FUNCTION_BLOCK PUBLIC VelocityCtrlAxis_FB
VAR_INPUT
	
	rAxisBasicFB 		: REFERENCE TO BasicAxis_FB ;
	rVelocityCtrl	 	: REFERENCE TO VelocityCtrl_typ ;
		
END_VAR

VAR_OUTPUT
END_VAR
	
VAR
	LogMsgInit		: BOOL;
	LogMsg_0 		: LogMsg ;
	
//	GetCycleTime:	FB_CTRL_GET_TASK_CYCLETIME;
//	CycleTime:		TIME;
//	CycleTimeInit:	BOOL;
	
	
	fbGetCurTaskIdx: 		GETCURTASKINDEX;
    TaskCycleTimeUDINT: 	UDINT;
    TaskCycleTime: 			TIME;

	EnableTrigger : Trigger ;
	
	DisableTriger	: Trigger ;
	Disable			: BOOL ;
	
// Change Oper params
	ChangeModeTrigger   : Trigger ;
	CngToVelocityState 	: SINT;
	PrevCngToVelocityState : SINT;
	// Change Oper params
	InitSctrlTrigger : Trigger ;
	InitSctrlState 	 : SINT;	

	
	ErrorTrig : Trigger ;
	AxisStep     : eVelocityCtrlState ;
	ReturnToAxisStep     : eVelocityCtrlState ;
	
	LastAxisStep : eVelocityCtrlState ;
	
	tmp_ErrorEntry			: Eh_ErrorEntry_typ;
	
	
	
	ReadPosCtrlParamDone 	: BOOL;	
	OldCyclicTorque 		: LREAL;		
	OldSctrlKp 				: LREAL;
	OldSctrlKi 				: LREAL;
	PrevVel 				: LREAL;
	Error					: BOOL;
	//Paramter
		
	CyclicTorqueAtPositionCtrl : LREAL;	
	

	
	Delay 			:	 TON;
	
	StartTestRead: BOOL;
	TestRead : BOOL;
END_VAR

// 
// At default set default torque
//
// Change mode to velocity control
// 
//
//
//
//
IF __ISVALIDREF( rAxisBasicFB) AND __ISVALIDREF(rVelocityCtrl) THEN
	
	

IF NOT LogMsgInit THEN 
	LogMsg_0.logData.category:=	rAxisBasicFB.AxisCtrlPtr^.Input.Parameter.ThreadName;     
	LogMsg_0.Enable:= 	TRUE; 	
END_IF

IF (TaskCycleTimeUDINT = 0) THEN
	fbGetCurTaskIdx();
	TaskCycleTimeUDINT := _TaskInfo[fbGetCurTaskIdx.index].CycleTime;
	TaskCycleTime	:= UDINT_TO_TIME(TaskCycleTimeUDINT/10000); 
END_IF



LogMsg_0.ptrGlobalArray:= 	ADR(LogGlobalArray);
LogMsg_0.ptrEncoderAngle:= 	ADR(rAxisBasicFB.AxisCtrlPtr^.Input.Parameter.PosForLog);



//in case of Stop go to STATE_WAIT
IF (rVelocityCtrl.Output.Status.Active)AND(NOT rVelocityCtrl.Output.Status.InStopVelCtrl)  THEN
	
	
	IF rAxisBasicFB.AxisCtrlPtr^.Output.Status.FAULT THEN
 
			AxisStep := eVelocityCtrlState.VELOCITY_CTRL_STATE_ERROR;	

	ELSIF (rAxisBasicFB.AxisCtrlPtr^.Input.Command.Halt) OR rVelocityCtrl.Input.Command.Stop THEN
		rVelocityCtrl.Input.Command.Stop := FALSE;
		Meth_stop(FALSE);
		AxisStep := eVelocityCtrlState.VELOCITY_CTRL_STATE_STOP ;

		
	ELSIF (rAxisBasicFB.AxisCtrlPtr^.Input.Command.Stop)  THEN 
		AxisStep := eVelocityCtrlState.VELOCITY_CTRL_ACTIVE_STAND_STILL;
		PrevVel :=  rVelocityCtrl.Input.Parameter.CyclicVelocity := 0;
	END_IF	
	
END_IF


IF EnableTrigger.EDGEPOS(rVelocityCtrl.Input.Command.Enable) THEN
 	IF (NOT rVelocityCtrl.Output.Status.Active) AND AxisStep = eVelocityCtrlState.VELOCITY_CTRL_STATE_READY THEN
		METH_ChangeToVelMode(FALSE);
		AxisStep := VELOCITY_CTRL_CNG_TO_VEL_MODE ;
	END_IF	
		
END_IF		
	
IF EnableTrigger.EDGENEG( rVelocityCtrl.Input.Command.Enable) THEN
	IF (rVelocityCtrl.Output.Status.Active) THEN
 		Meth_ExitVelCtrl(FALSE);
		AxisStep :=  eVelocityCtrlState.VELOCITY_CTRL_DISABLE;
	END_IF	
	
END_IF		



CASE AxisStep OF
		
	(******************** WAIT *************************)
		
	VELOCITY_CTRL_STATE_WAIT:	
		rVelocityCtrl.Output.Status.Active := FALSE;
		IF rAxisBasicFB.AxisCtrlPtr^.Output.Status.AxisInitDone
			 THEN
			AxisStep := VELOCITY_CTRL_STATE_READY ;
		END_IF
		
		THIS^.ResetAll_MC_FB();
		
	VELOCITY_CTRL_STATE_READY:
	
		rVelocityCtrl.Output.Status.Active := FALSE;
		IF rVelocityCtrl.Input.Command.InitSctrl THEN
				
				rVelocityCtrl.Input.Command.InitSctrl := FALSE;
				rVelocityCtrl.Output.Status.SctrlInitialized := FALSE;
				Meth_InitSctrl(FALSE);
				
				rAxisBasicFB.Meth_WriteObj(FALSE,enumMotionObject.VEL_KI,0);
				AxisStep :=VELOCITY_CTRL_InitSctrl;
				ReturnToAxisStep := VELOCITY_CTRL_STATE_READY;
 								
		ELSIF rVelocityCtrl.Input.Command.Stop THEN
			
			rVelocityCtrl.Input.Command.Stop  := FALSE;
			AxisStep := VELOCITY_CTRL_STATE_STOP ;
			
		ELSIF rVelocityCtrl.Input.Parameter.CyclicTorque <> OldCyclicTorque THEN
				
				Error := FALSE;
				ReturnToAxisStep := VELOCITY_CTRL_STATE_READY;
				AxisStep :=VELOCITY_CTRL_CHANGE_TORQUE;
				
				rAxisBasicFB.Meth_CngTorqueOffset(FALSE,0);
				rAxisBasicFB.Meth_CngMaxTorque(FALSE,0);
				ReturnToAxisStep := VELOCITY_CTRL_STATE_READY;
				rAxisBasicFB.Meth_WriteObj(FALSE,enumMotionObject.VEL_KI,0);	
				rVelocityCtrl.Output.Status.UpdateTorqueDone := FALSE;		
		END_IF
		

//ReadPosCtrlParamDone
		
	VELOCITY_CTRL_CNG_TO_VEL_MODE:
		// Change mode to velocity control
		IF METH_ChangeToVelMode(TRUE) THEN
			rVelocityCtrl.Output.Status.Active := TRUE;
			AxisStep :=VELOCITY_CTRL_MOVE_VELOCITY;
		END_IF	
			
	VELOCITY_CTRL_READ_POS_CTRL_VALUES:
			IF Meth_ReadPosCtrlValues(TRUE) THEN
				AxisStep :=VELOCITY_CTRL_MOVE_VELOCITY;
			END_IF
	
				
	VELOCITY_CTRL_MOVE_VELOCITY:
	
		IF rVelocityCtrl.Input.Parameter.CyclicVelocity <>0 OR rAxisBasicFB.AxisCtrlPtr^.Output.monitor.ActVelocity <>0  THEN
			Meth_MoveVel();
			AxisStep := VELOCITY_CTRL_WAIT_MOVE_VELOCITY_DONE;
		ELSE
			AxisStep := VELOCITY_CTRL_ACTIVE;
		END_IF	
	
	
	VELOCITY_CTRL_WAIT_MOVE_VELOCITY_DONE:	
		IF rAxisBasicFB.AxisCtrlPtr^.Output.Status.MC_MoveVelocity.In_Velocity THEN
			IF rVelocityCtrl.Input.Parameter.CyclicTorque <> 0 THEN
				Error := FALSE;
				ReturnToAxisStep := VELOCITY_CTRL_ACTIVE;
				AxisStep :=VELOCITY_CTRL_CHANGE_TORQUE;
				rAxisBasicFB.Meth_CngTorqueOffset(FALSE,0);
				rAxisBasicFB.Meth_CngMaxTorque(FALSE,0);
				ReturnToAxisStep := VELOCITY_CTRL_ACTIVE;
				rAxisBasicFB.Meth_WriteObj(FALSE,enumMotionObject.VEL_KI,0);
			ELSE
				PrevVel := rVelocityCtrl.Input.Parameter.CyclicVelocity;
				AxisStep := VELOCITY_CTRL_ACTIVE;
			END_IF	 
	END_IF
		
		
	VELOCITY_CTRL_ACTIVE:
	
			rVelocityCtrl.Output.Status.Active := TRUE;
			IF rVelocityCtrl.Input.Command.Stop THEN
				meth_Stop(FALSE);
				rVelocityCtrl.Input.Command.Stop  := FALSE;
				AxisStep := VELOCITY_CTRL_STATE_STOP ;
				
			ELSIF rVelocityCtrl.Input.Command.InitSctrl THEN
				
				rVelocityCtrl.Input.Command.InitSctrl := FALSE;
				rVelocityCtrl.Output.Status.SctrlInitialized := FALSE;
				Meth_InitSctrl(FALSE);
				
				rAxisBasicFB.Meth_WriteObj(FALSE,enumMotionObject.VEL_KI,0);
				AxisStep :=VELOCITY_CTRL_InitSctrl;
				ReturnToAxisStep := VELOCITY_CTRL_ACTIVE;
				
			ELSIF rVelocityCtrl.Input.Parameter.CyclicTorque <> OldCyclicTorque THEN
				
				Error := FALSE;
				ReturnToAxisStep := VELOCITY_CTRL_ACTIVE;
				AxisStep :=VELOCITY_CTRL_CHANGE_TORQUE;
				rAxisBasicFB.Meth_CngTorqueOffset(FALSE,0);
				rAxisBasicFB.Meth_CngMaxTorque(FALSE,0);
				ReturnToAxisStep := VELOCITY_CTRL_ACTIVE;
				rAxisBasicFB.Meth_WriteObj(FALSE,enumMotionObject.VEL_KI,0);				
			ELSIF rVelocityCtrl.Input.Parameter.CyclicVelocity <> rAxisBasicFB.AxisCtrlPtr^.Input.Parameter.Velocity THEN
					AxisStep := VELOCITY_CTRL_MOVE_VELOCITY;
		 	
			ELSIF rVelocityCtrl.Input.Parameter.CyclicVelocity <> PrevVel THEN
				
				AxisStep := VELOCITY_CTRL_MOVE_VELOCITY;
				
			END_IF	
			
	VELOCITY_CTRL_ACTIVE_STAND_STILL:
			rVelocityCtrl.Output.Status.Active := TRUE;
 			
			IF rVelocityCtrl.Input.Parameter.CyclicVelocity <> PrevVel THEN
				
				AxisStep := VELOCITY_CTRL_MOVE_VELOCITY;
			
			
			ELSIF rVelocityCtrl.Input.Command.InitSctrl THEN
				
				rVelocityCtrl.Input.Command.InitSctrl := FALSE;
				rVelocityCtrl.Output.Status.SctrlInitialized := FALSE;
				Meth_InitSctrl(FALSE);
				
				rAxisBasicFB.Meth_WriteObj(FALSE,enumMotionObject.VEL_KI,0);
				AxisStep :=VELOCITY_CTRL_InitSctrl;
				ReturnToAxisStep := VELOCITY_CTRL_ACTIVE_STAND_STILL;
				
			ELSIF rVelocityCtrl.Input.Parameter.CyclicTorque <> OldCyclicTorque THEN
				
				Error := FALSE;
				ReturnToAxisStep := VELOCITY_CTRL_ACTIVE;
				AxisStep :=VELOCITY_CTRL_CHANGE_TORQUE;
				rAxisBasicFB.Meth_CngTorqueOffset(FALSE,0);
				rAxisBasicFB.Meth_CngMaxTorque(FALSE,0);
				ReturnToAxisStep := VELOCITY_CTRL_ACTIVE_STAND_STILL;
				rAxisBasicFB.Meth_WriteObj(FALSE,enumMotionObject.VEL_KI,0);

		 	
			ELSIF rAxisBasicFB.AxisCtrlPtr^.Output.Status.AxisStatus.Coupled THEN
				IF rAxisBasicFB.AxisCtrlPtr^.Output.monitor.ActVelocity <> 0 THEN
					AxisStep := VELOCITY_CTRL_ACTIVE;
				END_IF 
			END_IF	

	VELOCITY_CTRL_InitSctrl:
	
			IF Meth_InitSctrl(TRUE,Error=>Error) THEN
				AxisStep :=ReturnToAxisStep;			
			END_IF
			
			IF Error THEN
			//	
			END_IF
	VELOCITY_CTRL_CHANGE_TORQUE:	
				
			IF rVelocityCtrl.Input.Parameter.TorqueMode = eTorqueMode.mcFF THEN
				//IF rAxisBasicFB.Meth_CngTorqueOffset(TRUE,rVelocityCtrl.Input.Parameter.CyclicTorque, Error => Error ) THEN
				IF  rAxisBasicFB.Meth_WriteObj(TRUE, enumMotionObject.TORQUE_OFFSET,rVelocityCtrl.Input.Parameter.CyclicTorque, Error => Error ) THEN
					fnLogMsg(ADR(LogMsg_0),LOG_INFO,'Vel Ctrl Change Torque to=%d',LREAL_TO_DINT(rVelocityCtrl.Input.Parameter.CyclicTorque*1000),0,0);
					
					OldCyclicTorque := rVelocityCtrl.Input.Parameter.CyclicTorque;
					rAxisBasicFB.Meth_CngTorqueOffset(FALSE,rVelocityCtrl.Input.Parameter.CyclicTorque);
					AxisStep :=ReturnToAxisStep;	
					rVelocityCtrl.Output.monitor.SetCyclicTorque := rVelocityCtrl.Input.Parameter.CyclicTorque ;
				END_IF							
			
			ELSIF rVelocityCtrl.Input.Parameter.TorqueMode = eTorqueMode.mcLimit THEN
				//IF rAxisBasicFB.Meth_CngMaxTorque(TRUE,rVelocityCtrl.Input.Parameter.CyclicTorque , Error => Error) THEN
				IF  rAxisBasicFB.Meth_WriteObj(TRUE, enumMotionObject.MAX_TORQUE,rVelocityCtrl.Input.Parameter.CyclicTorque, Error => Error ) THEN					
					OldCyclicTorque := rVelocityCtrl.Input.Parameter.CyclicTorque;
					rVelocityCtrl.Output.monitor.SetCyclicTorque := rVelocityCtrl.Input.Parameter.CyclicTorque ;
					rVelocityCtrl.Output.Status.UpdateTorqueDone := TRUE;
					AxisStep :=ReturnToAxisStep;
	
				END_IF
			END_IF
			
	eVelocityCtrlState.VELOCITY_CTRL_STATE_STOP:
		IF Meth_stop(TRUE) THEN
			
			PrevVel :=  rVelocityCtrl.Input.Parameter.CyclicVelocity := 0;
			AxisStep := eVelocityCtrlState.VELOCITY_CTRL_ACTIVE_STAND_STILL;
		END_IF
	
	
	eVelocityCtrlState.VELOCITY_CTRL_DISABLE:
		rVelocityCtrl.Output.Status.InStopVelCtrl := TRUE;
		IF Meth_ExitVelCtrl(TRUE) THEN
			rVelocityCtrl.Output.Status.InStopVelCtrl := FALSE;
			AxisStep := eVelocityCtrlState.VELOCITY_CTRL_STATE_READY;
		END_IF
	eVelocityCtrlState.VELOCITY_CTRL_STATE_RETURN_ORG_VALUES:
		IF Meth_ReturnOrgPosCtrlValues(TRUE) THEN				
			AxisStep := ReturnToAxisStep ;
		END_IF
		
	eVelocityCtrlState.VELOCITY_CTRL_STATE_ERROR:
			rVelocityCtrl.Output.Status.InStopVelCtrl := TRUE;
			IF Meth_ExitVelCtrl(TRUE) THEN			
				rVelocityCtrl.Output.Status.InStopVelCtrl := FALSE;
				AxisStep := eVelocityCtrlState.VELOCITY_CTRL_STATE_WAIT;
			END_IF

			

	
	
END_CASE 



//=====================================================================================================================\\

//IF CyclicAxisCtrlPtr^.Output.Error.ErrorID <> 0 THEN		
	//BasicAxisCtrlPtr^.Output.Error.ErrorID := CyclicAxisCtrlPtr^.Output.Error.ErrorID ;
	//CyclicAxisCtrlPtr^.Output.Error.ErrorID := 0;
//END_IF

	IF LastAxisStep <> AxisStep THEN
		
		fnLogMsg(ADR(LogMsg_0),LOG_INFO,'Vel Ctrl CurSt=%d LstSt=%d',AxisStep,LastAxisStep,0);
		LastAxisStep := AxisStep ;
	END_IF	
	
	IF StartTestRead THEN
		StartTestRead := FALSE;
		Meth_ReadPosCtrlValues(FALSE);
		TestRead := TRUE;
		
	ELSIF TestRead THEN
		IF Meth_ReadPosCtrlValues(TRUE) THEN
			TestRead := FALSE;
		END_IF	
		
	END_IF

	
	
//fnLogTransfer FUNCTION call
fnLogTransfer(ADR(LogMsg_0));
		

END_IF

METHOD AddNCError : BOOL
VAR_INPUT
	ErrorId			: UDINT;
	ErrorPrefix     : STRING[100];
END_VAR

	tmp_ErrorEntry.ErrorId		:= ErrorId;

	tmp_ErrorEntry.ErrorText	:= ErrorPrefix;

	tmp_ErrorEntry.ErrorText	:= CONCAT(tmp_ErrorEntry.ErrorText, UDINT_TO_STRING(tmp_ErrorEntry.ErrorId));
	tmp_ErrorEntry.ErrorText	:= CONCAT(tmp_ErrorEntry.ErrorText, 'Task: ');
	tmp_ErrorEntry.ErrorText	:= CONCAT(tmp_ErrorEntry.ErrorText, rVelocityCtrl.Input.Parameter.ThreadName);	
	tmp_ErrorEntry.ErrorText	:= CONCAT(tmp_ErrorEntry.ErrorText, FC_NcErrorMsg(tmp_ErrorEntry.ErrorId));	
	fnLogMsg(ADR(LogMsg_0),LOG_ERROR,tmp_ErrorEntry.ErrorText,0,0,0);	
	
	tmp_ErrorEntry.MotorEvents := CreateNCErrMsgDetails(tmp_ErrorEntry.ErrorId);
	
	rAxisBasicFB.AxisCtrlPtr^.Output.Error.fbErrorHandler.ErrorPush(tmp_ErrorEntry);
END_METHOD

METHOD METH_ChangeToVelMode : BOOL
VAR_INPUT
	Execute : BOOL;
END_VAR
VAR_INST
	DelayBeforeChangimeMode: TON;
END_VAR
IF InitSctrlTrigger.EDGEPOS( Execute) THEN
	CngToVelocityState := 1;
	METH_ChangeToVelMode := FALSE;
	rAxisBasicFB.AxisCtrlPtr^.Input.Command.Power := FALSE;
	
	OldCyclicTorque := 0;		
	OldSctrlKp 		:= 0;
	OldSctrlKi 		:= 0;			
	rAxisBasicFB.Meth_WriteObj (FALSE, enumMotionobject.OPERATION_MODE,DINT_TO_LREAL(eDriveModeOfOperation.CyclicSyncVelocity));

END_IF

IF InitSctrlTrigger.EDGENEG( Execute) THEN
	CngToVelocityState := 0;
END_IF


CASE CngToVelocityState OF
	0:
		METH_ChangeToVelMode := FALSE;
		 
	1:
		DelayBeforeChangimeMode.IN := FALSE;
		IF ReadPosCtrlParamDone = FALSE THEN
			 Meth_ReadPosCtrlValues(FALSE);
			 CngToVelocityState := CngToVelocityState +1;	
		ELSE
			CngToVelocityState := CngToVelocityState +2;
		END_IF		
	2:
		IF Meth_ReadPosCtrlValues(TRUE) THEN
			
			rAxisBasicFB.Meth_WriteObj (FALSE, enumMotionobject.OPERATION_MODE,eDriveModeOfOperation.CyclicSyncVelocity);
			
			CngToVelocityState := CngToVelocityState +1;
			
		END_IF
	3:	//Change mode to velocity control
		IF rAxisBasicFB.Meth_WriteObj (TRUE, enumMotionobject.OPERATION_MODE,eDriveModeOfOperation.CyclicSyncVelocity) THEN			
			rAxisBasicFB.Meth_WriteObj (FALSE, enumMotionobject.OPERATION_MODE,eDriveModeOfOperation.CyclicSyncVelocity);
			CngToVelocityState := CngToVelocityState +1;
		END_IF
		
	4://Disable Gain Control
		IF NOT rAxisBasicFB.AxisCtrlPtr^.Output.Status.MC_Power.Status THEN
			IF rAxisBasicFB.Meth_WriteObj (TRUE, enumMotionobject.GAIN_SCHEDULE,0) THEN			
				rAxisBasicFB.Meth_WriteObj (FALSE, enumMotionobject.OPERATION_MODE,eDriveModeOfOperation.CyclicSyncVelocity);			
				CngToVelocityState := CngToVelocityState +1;
			END_IF
		END_IF	
	
	5:	
		DelayBeforeChangimeMode.IN := TRUE;
		DelayBeforeChangimeMode.PT := T#10S;
		IF DelayBeforeChangimeMode.Q THEN
			rAxisBasicFB.AxisCtrlPtr^.Input.Command.Power := TRUE;
			IF rAxisBasicFB.AxisCtrlPtr^.Output.Status.AxisStatus.StandStill THEN
				CngToVelocityState := CngToVelocityState +1;
			END_IF
		END_IF	
	6:
		IF  rAxisBasicFB.Meth_WriteObj(TRUE, enumMotionObject.ACC_CLOSE_POS_ERR ,   rVelocityCtrl.Input.Parameter.CyclicVelocity    , Error =>Error ) THEN
			rAxisBasicFB.Meth_WriteObj(FALSE, enumMotionObject.ACC_CLOSE_POS_ERR ,0 );
			CngToVelocityState := CngToVelocityState +1;
		END_IF	
	
	7:	
		METH_ChangeToVelMode := TRUE;
END_CASE

DelayBeforeChangimeMode();

	IF CngToVelocityState <> PrevCngToVelocityState THEN
		
		fnLogMsg(ADR(LogMsg_0),LOG_INFO,'CngToVelocityState CurSt=%d LstSt=%d',CngToVelocityState,PrevCngToVelocityState,0);
		PrevCngToVelocityState := CngToVelocityState ;
	END_IF
END_METHOD

METHOD Meth_ExitVelCtrl : BOOL
VAR_INPUT
	Execute   : BOOL;
END_VAR

VAR_INST
	// Service Functions Variablea
	StopTrigger : Trigger ;
	ExitState  		 : SINT;
	PrevExitState   : SINT;
END_VAR

VAR_OUTPUT
	Error : BOOL;
END_VAR

IF StopTrigger.EDGEPOS(Execute) THEN
	ExitState  := 1;
	Meth_ExitVelCtrl := FALSE;
 	Meth_ReturnOrgPosCtrlValues(FALSE) ;
	Error := FALSE;
END_IF


IF StopTrigger.EDGENEG(Execute) THEN
	 PrevExitState := 0;
	 ExitState:= 0;
END_IF


CASE ExitState OF
	 		
	
	1:	 
		
//			
 //  	
		Delay(IN:=	FALSE);
		IF rAxisBasicFB.AxisCtrlPtr^.Output.Status.AxisStatus.StandStill = FALSE  AND rAxisBasicFB.AxisCtrlPtr^.Output.Status.AxisStatus.Disabled = FALSE THEN
		//	rAxisBasicFB.AxisCtrlPtr^.Input.Command.MoveVelocity := TRUE;	
		//	rAxisBasicFB.AxisCtrlPtr^.Input.Parameter.Velocity   := 100;
			rAxisBasicFB.AxisCtrlPtr^.Input.Command.Stop := TRUE;		
			ExitState := ExitState +1;
		ELSE
			ExitState := 3;
		END_IF	
					
   						
		
		
		
	2:
			IF (rAxisBasicFB.AxisCtrlPtr^.Output.Status.AxisStatus.StandStill OR rAxisBasicFB.AxisCtrlPtr^.Output.Status.AxisStatus.Disabled)				
			//IF rAxisBasicFB.AxisCtrlPtr^.Output.Status.MC_MoveVelocity.In_Velocity 
				 THEN
				Delay.PT := T#2S;
				Delay(IN:=	TRUE);
				IF Delay.Q THEN
					ExitState := ExitState +1;
				END_IF								
			END_IF

	
	3:
			rAxisBasicFB.AxisCtrlPtr^.Input.Command.Power := FALSE;

			ExitState := ExitState +1;

	4:
		IF rAxisBasicFB.AxisCtrlPtr^.Output.Status.AxisStatus.Disabled THEN
			IF ReadPosCtrlParamDone THEN
				IF  rAxisBasicFB.Meth_WriteObj(TRUE, enumMotionObject.ACC_CLOSE_POS_ERR ,  rVelocityCtrl.Output.monitor.OrgAccToCloseThePosError, Error =>Error ) THEN
					rAxisBasicFB.Meth_WriteObj(FALSE, enumMotionObject.ACC_CLOSE_POS_ERR ,0 );
					ExitState := ExitState +1;
				END_IF
			ELSE	
				ExitState := ExitState +1;
			END_IF
			
		END_IF	
	

	5:
		IF ReadPosCtrlParamDone THEN
			IF Meth_ReturnOrgPosCtrlValues(TRUE) THEN
				ExitState := ExitState +1;
			END_IF
		ELSE	
			ExitState := ExitState +1;
		END_IF
	
	
	6:		
		IF rAxisBasicFB.Meth_WriteObj (TRUE, enumMotionobject.OPERATION_MODE,TO_LREAL(eDriveModeOfOperation.CyclicSyncMode)) THEN
			rAxisBasicFB.Meth_WriteObj (FALSE, enumMotionobject.OPERATION_MODE,0);
			Delay.IN := FALSE;
			ExitState := ExitState +1;
		END_IF
	7:
			Delay.IN := TRUE;
			Delay.PT := T#2S;
			Delay();
			IF Delay.Q THEN
				ExitState := ExitState +1;
				Delay.IN := FALSE;
			END_IF

	8:
 		Meth_ExitVelCtrl := TRUE;
		

	

END_CASE

	IF ExitState <> PrevExitState THEN
		
		fnLogMsg(ADR(LogMsg_0),LOG_INFO,'Exit Vel Ctrl CurSt=%d LstSt=%d',ExitState,PrevExitState,0);
		PrevExitState := ExitState ;
	END_IF
END_METHOD

METHOD Meth_InitSctrl : BOOL
VAR_INPUT
	Execute : BOOL;
END_VAR


VAR_OUTPUT
	Error : BOOL;
END_VAR
IF InitSctrlTrigger.EDGEPOS(Execute) THEN
	InitSctrlState  := 1;
	Meth_InitSctrl := FALSE;
	rAxisBasicFB.Meth_InitVelKP (FALSE,0);
	rAxisBasicFB.Meth_InitVelKI(FALSE,0);
	Error := FALSE;
END_IF


IF InitSctrlTrigger.EDGENEG(Execute) THEN
	
	 InitSctrlState:= 0;
END_IF


CASE InitSctrlState OF
	 
		
	1:
		 			
			IF rAxisBasicFB.Meth_InitVelKP (TRUE,(rVelocityCtrl.Input.Parameter.SctrlKp), Error=>Error) THEN
				OldSctrlKp := rVelocityCtrl.Input.Parameter.SctrlKp;
				InitSctrlState := InitSctrlState +1;
				rAxisBasicFB.Meth_InitVelKP (FALSE,rVelocityCtrl.Input.Parameter.SctrlKp);
			END_IF	
  
			

	2:
	
		IF rAxisBasicFB.Meth_InitVelKI(TRUE,(rVelocityCtrl.Input.Parameter.SctrlKi), Error=>Error) THEN
			rAxisBasicFB.Meth_InitVelKP (FALSE,rVelocityCtrl.Input.Parameter.SctrlKi);
			OldSctrlKi := rVelocityCtrl.Input.Parameter.SctrlKi ;
			InitSctrlState := InitSctrlState +1;
		END_IF	

		IF Error THEN
		//	
		END_IF
		
	3:		
		rAxisBasicFB.Meth_WriteObj(FALSE,enumMotionObject.VEL_KI,0);
		rVelocityCtrl.Output.Status.SctrlInitialized := TRUE;
		Meth_InitSctrl := TRUE; 
	END_CASE
END_METHOD

METHOD Meth_MoveVel : BOOL
VAR_INPUT
END_VAR
	rAxisBasicFB.AxisCtrlPtr^.Input.Parameter.Velocity 	   := rVelocityCtrl.Input.Parameter.CyclicVelocity;
	rAxisBasicFB.AxisCtrlPtr^.Input.Parameter.Acceleration := rVelocityCtrl.Input.Parameter.Acceleration;
	rAxisBasicFB.AxisCtrlPtr^.Input.Parameter.Deceleration := rVelocityCtrl.Input.Parameter.Deceleration;
	
	rAxisBasicFB.AxisCtrlPtr^.Input.Command.MoveVelocity := TRUE;
END_METHOD

METHOD Meth_ReadPosCtrlValues : BOOL
VAR_INPUT
	Execute : BOOL;
END_VAR


VAR_INST
	// Service Functions Variablea
		 
	ReadOrginalValuesTrigger : Trigger ;
	ReadOrginalValuesState   : SINT;
END_VAR	

VAR_OUTPUT
	Error : BOOL;	
END_VAR
IF ReadOrginalValuesTrigger.EDGEPOS(Execute) THEN
	ReadOrginalValuesState  := 1;
	Meth_ReadPosCtrlValues := FALSE;
	Error := FALSE;
	rAxisBasicFB.Meth_ReadObj(FALSE, enumMotionObject.MAX_TORQUE, Value =>rVelocityCtrl.Output.monitor.OrgMaxTorque, Error =>Error );
END_IF


IF ReadOrginalValuesTrigger.EDGENEG(Execute) THEN
	 rAxisBasicFB.Meth_ReadObj(FALSE, enumMotionObject.MAX_TORQUE, Value =>rVelocityCtrl.Output.monitor.OrgMaxTorque, Error =>Error );
	 ReadOrginalValuesState:= 0;
END_IF


CASE ReadOrginalValuesState OF
	 
		
	1:
		IF  rAxisBasicFB.Meth_ReadObj(TRUE, enumMotionObject.TORQUE_OFFSET, Value =>rVelocityCtrl.Output.monitor.OrgCyclicTorque, Error =>Error ) THEN
			fnLogMsg(ADR(LogMsg_0),LOG_INFO,'TORQUE_OFFSET org=%d',TO_DINT(rVelocityCtrl.Output.monitor.OrgCyclicTorque),0,0);
			rAxisBasicFB.Meth_ReadObj(FALSE, enumMotionObject.TORQUE_OFFSET  );
 			ReadOrginalValuesState := ReadOrginalValuesState +1;
			Error := FALSE;						
		END_IF
		IF Error THEN
			ReadOrginalValuesState := 33;
		END_IF
			
	2:
		IF  rAxisBasicFB.Meth_ReadObj(TRUE, enumMotionObject.VEL_KP, Value =>rVelocityCtrl.Output.monitor.OrgSctrlKp, Error =>Error ) THEN
			rVelocityCtrl.Output.monitor.OrgVelKp := rVelocityCtrl.Output.monitor.OrgSctrlKp;
			
			fnLogMsg(ADR(LogMsg_0),LOG_INFO,'VEL_KP org=%d',TO_DINT(rVelocityCtrl.Output.monitor.OrgSctrlKp),0,0);
			rAxisBasicFB.Meth_ReadObj(FALSE, enumMotionObject.TORQUE_OFFSET  );
 			ReadOrginalValuesState := ReadOrginalValuesState +1;
		END_IF
	3:
		IF  rAxisBasicFB.Meth_ReadObj(TRUE, enumMotionObject.VEL_KI, Value =>rVelocityCtrl.Output.monitor.OrgSctrlKi, Error =>Error ) THEN
			fnLogMsg(ADR(LogMsg_0),LOG_INFO,'VEL_KI org=%d',TO_DINT(rVelocityCtrl.Output.monitor.OrgSctrlKi),0,0);
			rAxisBasicFB.Meth_ReadObj(FALSE, enumMotionObject.TORQUE_OFFSET  );
 			ReadOrginalValuesState := ReadOrginalValuesState +1;
		END_IF
	
	4:
		IF rAxisBasicFB.Meth_ReadObj (TRUE, enumMotionobject.GAIN_SCHEDULE, Value =>rVelocityCtrl.Output.monitor.OrgGainCtrl, Error =>Error) THEN
				fnLogMsg(ADR(LogMsg_0),LOG_INFO,'GAIN_SCHEDULE org=%d',TO_DINT(rVelocityCtrl.Output.monitor.OrgGainCtrl),0,0);			
				rAxisBasicFB.Meth_ReadObj(FALSE, enumMotionObject.TORQUE_OFFSET  );
				ReadOrginalValuesState := ReadOrginalValuesState +1;						
		END_IF		
		
	5:
	

			IF rAxisBasicFB.Meth_ReadObj (TRUE, enumMotionobject.ACC_CLOSE_POS_ERR, Value =>rVelocityCtrl.Output.monitor.OrgAccToCloseThePosError, Error =>Error) THEN
				fnLogMsg(ADR(LogMsg_0),LOG_INFO,'ACC_CLOSE_POS_ERR org=%d',TO_DINT(rVelocityCtrl.Output.monitor.OrgAccToCloseThePosError),0,0);			
				rAxisBasicFB.Meth_ReadObj(FALSE, enumMotionObject.TORQUE_OFFSET  );
				ReadOrginalValuesState := ReadOrginalValuesState +1;						
			END_IF		

	7:		
		ReadPosCtrlParamDone := TRUE;
		Meth_ReadPosCtrlValues := TRUE; 
	END_CASE
END_METHOD

METHOD Meth_ReturnOrgPosCtrlValues : BOOL
VAR_INPUT
	Execute : BOOL;
END_VAR


VAR_INST
	// Service Functions Variablea
	ReturnOrginalTrigger : Trigger ;
	ReturnOrginalState   : SINT;
END_VAR	

VAR_OUTPUT
	Error : BOOL;
END_VAR
IF ReturnOrginalTrigger.EDGEPOS(Execute) THEN
	ReturnOrginalState  := 1;
	Meth_ReturnOrgPosCtrlValues := FALSE;
	Error := FALSE;
	rAxisBasicFB.Meth_WriteObj(FALSE, enumMotionObject.MAX_TORQUE, rVelocityCtrl.Output.monitor.OrgMaxTorque, Error =>Error );
	fnLogMsg(ADR(LogMsg_0),LOG_INFO,'VelCtrl Start Return Org Values',0,0,0);
END_IF


IF ReturnOrginalTrigger.EDGENEG(Execute) THEN
	 rAxisBasicFB.Meth_WriteObj(FALSE, enumMotionObject.MAX_TORQUE,  rVelocityCtrl.Output.monitor.OrgMaxTorque, Error =>Error );
	 ReturnOrginalState:= 0;
END_IF


CASE ReturnOrginalState OF
	 
		
	1:	
		IF  rAxisBasicFB.Meth_WriteObj(TRUE, enumMotionObject.GAIN_SCHEDULE,  rVelocityCtrl.Output.monitor.OrgGainCtrl, Error =>Error ) THEN
			rAxisBasicFB.Meth_WriteObj(FALSE, enumMotionObject.GAIN_SCHEDULE ,0 );
 			ReturnOrginalState := ReturnOrginalState +1;
		END_IF		
			
	2:
		IF  rAxisBasicFB.Meth_WriteObj(TRUE, enumMotionObject.VEL_KP,  rVelocityCtrl.Output.monitor.OrgSctrlKp, Error =>Error ) THEN
			rAxisBasicFB.Meth_WriteObj(FALSE,enumMotionObject.VEL_KP,0  );
 			ReturnOrginalState := ReturnOrginalState +1;
		END_IF
	3:
		IF  rAxisBasicFB.Meth_WriteObj(TRUE, enumMotionObject.VEL_KI,  rVelocityCtrl.Output.monitor.OrgSctrlKi, Error =>Error ) THEN
			rAxisBasicFB.Meth_WriteObj(FALSE, enumMotionObject.VEL_KP ,0 );
 			ReturnOrginalState := ReturnOrginalState +1;
		END_IF
	
	4:
		IF  rAxisBasicFB.Meth_WriteObj(TRUE, enumMotionObject.TORQUE_OFFSET, rVelocityCtrl.Output.monitor.OrgCyclicTorque , Error =>Error ) THEN
			rAxisBasicFB.Meth_WriteObj(FALSE, enumMotionObject.VEL_KP ,0 );
 			ReturnOrginalState := ReturnOrginalState +1;
		END_IF
		
	5:
	
	        IF rAxisBasicFB.Meth_WriteObj(TRUE, enumMotionObject.MAX_TORQUE,rVelocityCtrl.Output.monitor.OrgMaxTorque   , Error =>Error ) THEN	
				rAxisBasicFB.Meth_WriteObj(FALSE, enumMotionObject.VEL_KP ,0 );									
				rAxisBasicFB.Meth_WriteObj(FALSE, enumMotionObject.VEL_KP ,0 );
				ReturnOrginalState := ReturnOrginalState +1;					
			END_IF	
	
	6:			
		fnLogMsg(ADR(LogMsg_0),LOG_INFO,'VelCtrl Return Org Values Done',0,0,0);
		Meth_ReturnOrgPosCtrlValues := TRUE; 
	END_CASE
END_METHOD

METHOD Meth_Stop : BOOL
VAR_INPUT
	Execute   : BOOL;
END_VAR

VAR_INST
	// Service Functions Variablea
	StopTrigger : Trigger ;
	StopState   : SINT;
	
END_VAR

VAR_OUTPUT
	Error : BOOL;
END_VAR

IF StopTrigger.EDGEPOS(Execute) THEN
	StopState  := 1;
	Meth_Stop := FALSE;
 	Meth_ReturnOrgPosCtrlValues(FALSE) ;
	Error := FALSE;
END_IF


IF StopTrigger.EDGENEG(Execute) THEN
	
	 StopState:= 0;
END_IF


CASE StopState OF
 		
	
	1:	 
		
		rAxisBasicFB.AxisCtrlPtr^.Input.Command.Stop := TRUE;			
   		StopState := StopState +1;				
		Delay(IN:=	FALSE);
		
	2:
			IF rAxisBasicFB.AxisCtrlPtr^.Output.Status.AxisStatus.StandStill OR rAxisBasicFB.AxisCtrlPtr^.Output.Status.AxisStatus.Disabled THEN
				StopState := StopState +1;								
			END_IF

	


	3:
 		Meth_Stop := TRUE;
		

	

END_CASE
END_METHOD

METHOD PRIVATE ResetAll_MC_FB : BOOL
VAR_INPUT
END_VAR

		ResetAll_MC_FB := FALSE ;
				

		{warning disable C0371}
		//Warning: Access to VAR_IN_OUT <Var> declared in <POU> from external context <Method/Transition/Property>

		{warning restore C0371}
		
		
		memset(ADR(rVelocityCtrl.Input.Command) ,0 ,SIZEOF(rVelocityCtrl.Input.Command));
		memset(ADR(rVelocityCtrl.Output.Status) ,0 ,SIZEOF(rVelocityCtrl.Output.Status));
		
		ResetAll_MC_FB := TRUE ;
END_METHOD

END_FUNCTION_BLOCK

(* stored: Version 1.1.0.1, ProductVersion 3.1.4024.3
   POU VelocityCtrlAxis_FB: Id {19370e93-5365-40c7-98c2-dbdaeb676dae}, SpecialFunc None
   Method AddNCError: Id {488d80fa-883c-426c-914b-bb08d3f436f8}
   Method METH_ChangeToVelMode: Id {8d3c00e6-2673-423e-a136-0e9b875dc2a9}
   Method Meth_ExitVelCtrl: Id {146a8395-1da9-41a8-a600-93647740d164}
   Method Meth_InitSctrl: Id {277293a0-46b0-40c8-8c25-a830667691a3}
   Method Meth_MoveVel: Id {fa95af4a-6066-43df-ac87-41e58c9d8e8e}
   Method Meth_ReadPosCtrlValues: Id {4522cc7f-b585-4b24-8d4a-c04a901aa0ce}
   Method Meth_ReturnOrgPosCtrlValues: Id {3131fbc1-9b26-46ab-a59b-b748e02e062b}
   Method Meth_Stop: Id {98e371b4-4151-4e06-920d-8aeecd31293a}
   Method ResetAll_MC_FB: Id {64befd56-77af-467d-b520-45554e5bcca0} *)
